// TwinCAT 3 PLC project PLC
// Title: Test
// Company: Gema
// Author: RG
// ProjectVersion: 0.1.0.0
// ProgramVersion: 3.1.4023.0
// libraries:
//   Tc2_EtherCAT, * (Beckhoff Automation GmbH)
//   Tc2_Standard, * (Beckhoff Automation GmbH)
//   Tc2_System, * (Beckhoff Automation GmbH)
//   Tc3_Module, * (Beckhoff Automation GmbH)
//   TcoCore, 0.11.0.15 (Vortex.Library)
//   TcoData, 0.11.0.15 (Vortex.Library)
//   TcoDrivesBeckhoff, 0.11.0.15 (Vortex.Library)
//   TcoElements, 0.11.0.15 (Vortex.Library)
//   TcoPneumatics, 0.11.0.15 (Vortex.Library)
//   Vision.Library, * (Gema Technik)
//   BASIC,3.31,OSCAT
// project tree:
//   / PlcTask.TcTTO (not stored)
//   POUs/ AppContext.TcPOU (not stored), MAIN.TcPOU (not stored), MainStation.TcPOU
// real-time tasks:
//   TASK PlcTask: cycle T#1ms, priority 20, ADS port 350
// I/O:
//   DEVICE Device 2 (EtherCAT), AmsNetId 192.168.1.8.3.1
//     Box 1 (DL-EC1A) [DL-EC1A]
// variable links:
//   PLC/PLC Instance <-> Device 2 (EtherCAT)/Box 1 (DL-EC1A)
//     PlcTask Inputs/MAIN._app._mainStation._IvController.ID01 <-> ID01 Current Value  TxPDOMap/ID01 Current Value (P.V.)
//     PlcTask Inputs/MAIN._app._mainStation._IvController.ID01Status @bit 9 <-> ID01 Status TxPDOMap/ID01 Current Value Invalid
//     PlcTask Inputs/MAIN._app._mainStation._IvController.ID02Status @bit 9 <-> ID02 Status TxPDOMap/ID02 Current Value Invalid
//     PlcTask Inputs/MAIN._app._mainStation._IvController.ID03Status @bit 9 <-> ID03 Status TxPDOMap/ID03 Current Value Invalid
//     PlcTask Inputs/MAIN._app._mainStation._IvController.ID04Status @bit 9 <-> ID04 Status TxPDOMap/ID04 Current Value Invalid
//     PlcTask Inputs/MAIN._app._mainStation._IvController.ID05Status @bit 9 <-> ID05 Status TxPDOMap/ID05 Current Value Invalid
//     PlcTask Inputs/MAIN._app._mainStation._IvController.ID06Status @bit 9 <-> ID06 Status TxPDOMap/ID06 Current Value Invalid
//     PlcTask Inputs/MAIN._app._mainStation._IvController.ID07Status @bit 9 <-> ID07 Status TxPDOMap/ID07 Current Value Invalid
//     PlcTask Inputs/MAIN._app._mainStation._IvController.ID08Status @bit 9 <-> ID08 Status TxPDOMap/ID08 Current Value Invalid
//     PlcTask Inputs/MAIN._app._mainStation._IvController.ID01Status @bit 11 <-> ID01 Status TxPDOMap/ID01 Current Value Over Range
//     PlcTask Inputs/MAIN._app._mainStation._IvController.ID02Status @bit 11 <-> ID02 Status TxPDOMap/ID02 Current Value Over Range
//     PlcTask Inputs/MAIN._app._mainStation._IvController.ID03Status @bit 11 <-> ID03 Status TxPDOMap/ID03 Current Value Over Range
//     PlcTask Inputs/MAIN._app._mainStation._IvController.ID04Status @bit 11 <-> ID04 Status TxPDOMap/ID04 Current Value Over Range
//     PlcTask Inputs/MAIN._app._mainStation._IvController.ID05Status @bit 11 <-> ID05 Status TxPDOMap/ID05 Current Value Over Range
//     PlcTask Inputs/MAIN._app._mainStation._IvController.ID06Status @bit 11 <-> ID06 Status TxPDOMap/ID06 Current Value Over Range
//     PlcTask Inputs/MAIN._app._mainStation._IvController.ID07Status @bit 11 <-> ID07 Status TxPDOMap/ID07 Current Value Over Range
//     PlcTask Inputs/MAIN._app._mainStation._IvController.ID08Status @bit 11 <-> ID08 Status TxPDOMap/ID08 Current Value Over Range
//     PlcTask Inputs/MAIN._app._mainStation._IvController.ID01Status @bit 10 <-> ID01 Status TxPDOMap/ID01 Current Value Under Range
//     PlcTask Inputs/MAIN._app._mainStation._IvController.ID02Status @bit 10 <-> ID02 Status TxPDOMap/ID02 Current Value Under Range
//     PlcTask Inputs/MAIN._app._mainStation._IvController.ID03Status @bit 10 <-> ID03 Status TxPDOMap/ID03 Current Value Under Range
//     PlcTask Inputs/MAIN._app._mainStation._IvController.ID04Status @bit 10 <-> ID04 Status TxPDOMap/ID04 Current Value Under Range
//     PlcTask Inputs/MAIN._app._mainStation._IvController.ID05Status @bit 10 <-> ID05 Status TxPDOMap/ID05 Current Value Under Range
//     PlcTask Inputs/MAIN._app._mainStation._IvController.ID06Status @bit 10 <-> ID06 Status TxPDOMap/ID06 Current Value Under Range
//     PlcTask Inputs/MAIN._app._mainStation._IvController.ID07Status @bit 10 <-> ID07 Status TxPDOMap/ID07 Current Value Under Range
//     PlcTask Inputs/MAIN._app._mainStation._IvController.ID08Status @bit 10 <-> ID08 Status TxPDOMap/ID08 Current Value Under Range
//     PlcTask Inputs/MAIN._app._mainStation._IvController.ID01Status @bit 15 <-> ID01 Status TxPDOMap/ID01 Error Status
//     PlcTask Inputs/MAIN._app._mainStation._IvController.ID02Status @bit 15 <-> ID02 Status TxPDOMap/ID02 Error Status
//     PlcTask Inputs/MAIN._app._mainStation._IvController.ID03Status @bit 15 <-> ID03 Status TxPDOMap/ID03 Error Status
//     PlcTask Inputs/MAIN._app._mainStation._IvController.ID04Status @bit 15 <-> ID04 Status TxPDOMap/ID04 Error Status
//     PlcTask Inputs/MAIN._app._mainStation._IvController.ID05Status @bit 15 <-> ID05 Status TxPDOMap/ID05 Error Status
//     PlcTask Inputs/MAIN._app._mainStation._IvController.ID06Status @bit 15 <-> ID06 Status TxPDOMap/ID06 Error Status
//     PlcTask Inputs/MAIN._app._mainStation._IvController.ID07Status @bit 15 <-> ID07 Status TxPDOMap/ID07 Error Status
//     PlcTask Inputs/MAIN._app._mainStation._IvController.ID08Status @bit 15 <-> ID08 Status TxPDOMap/ID08 Error Status
//     PlcTask Inputs/MAIN._app._mainStation._IvController.ID01Status <-> ID01 Status TxPDOMap/ID01 Output 1
//     PlcTask Inputs/MAIN._app._mainStation._IvController.ID02Status <-> ID02 Status TxPDOMap/ID02 Output 1
//     PlcTask Inputs/MAIN._app._mainStation._IvController.ID03Status <-> ID03 Status TxPDOMap/ID03 Output 1
//     PlcTask Inputs/MAIN._app._mainStation._IvController.ID04Status <-> ID04 Status TxPDOMap/ID04 Output 1
//     PlcTask Inputs/MAIN._app._mainStation._IvController.ID05Status <-> ID05 Status TxPDOMap/ID05 Output 1
//     PlcTask Inputs/MAIN._app._mainStation._IvController.ID06Status <-> ID06 Status TxPDOMap/ID06 Output 1
//     PlcTask Inputs/MAIN._app._mainStation._IvController.ID07Status <-> ID07 Status TxPDOMap/ID07 Output 1
//     PlcTask Inputs/MAIN._app._mainStation._IvController.ID08Status <-> ID08 Status TxPDOMap/ID08 Output 1
//     PlcTask Inputs/MAIN._app._mainStation._IvController.ID01Status @bit 1 <-> ID01 Status TxPDOMap/ID01 Output 2
//     PlcTask Inputs/MAIN._app._mainStation._IvController.ID01Status @bit 2 <-> ID01 Status TxPDOMap/ID01 Output 3
//     PlcTask Inputs/MAIN._app._mainStation._IvController.ID01Status @bit 3 <-> ID01 Status TxPDOMap/ID01 Output 4
//     PlcTask Inputs/MAIN._app._mainStation._IvController.ID01Status @bit 4 <-> ID01 Status TxPDOMap/ID01 Output 5
//     PlcTask Inputs/MAIN._app._mainStation._IvController.ID02Status @bit 1 <-> ID02 Status TxPDOMap/ID02 Output 2
//     PlcTask Inputs/MAIN._app._mainStation._IvController.ID02Status @bit 2 <-> ID02 Status TxPDOMap/ID02 Output 3
//     PlcTask Inputs/MAIN._app._mainStation._IvController.ID02Status @bit 3 <-> ID02 Status TxPDOMap/ID02 Output 4
//     PlcTask Inputs/MAIN._app._mainStation._IvController.ID02Status @bit 4 <-> ID02 Status TxPDOMap/ID02 Output 5
//     PlcTask Inputs/MAIN._app._mainStation._IvController.ID03Status @bit 1 <-> ID03 Status TxPDOMap/ID03 Output 2
//     PlcTask Inputs/MAIN._app._mainStation._IvController.ID03Status @bit 2 <-> ID03 Status TxPDOMap/ID03 Output 3
//     PlcTask Inputs/MAIN._app._mainStation._IvController.ID03Status @bit 3 <-> ID03 Status TxPDOMap/ID03 Output 4
//     PlcTask Inputs/MAIN._app._mainStation._IvController.ID03Status @bit 4 <-> ID03 Status TxPDOMap/ID03 Output 5
//     PlcTask Inputs/MAIN._app._mainStation._IvController.ID04Status @bit 1 <-> ID04 Status TxPDOMap/ID04 Output 2
//     PlcTask Inputs/MAIN._app._mainStation._IvController.ID04Status @bit 2 <-> ID04 Status TxPDOMap/ID04 Output 3
//     PlcTask Inputs/MAIN._app._mainStation._IvController.ID04Status @bit 3 <-> ID04 Status TxPDOMap/ID04 Output 4
//     PlcTask Inputs/MAIN._app._mainStation._IvController.ID04Status @bit 4 <-> ID04 Status TxPDOMap/ID04 Output 5
//     PlcTask Inputs/MAIN._app._mainStation._IvController.ID05Status @bit 1 <-> ID05 Status TxPDOMap/ID05 Output 2
//     PlcTask Inputs/MAIN._app._mainStation._IvController.ID05Status @bit 2 <-> ID05 Status TxPDOMap/ID05 Output 3
//     PlcTask Inputs/MAIN._app._mainStation._IvController.ID05Status @bit 3 <-> ID05 Status TxPDOMap/ID05 Output 4
//     PlcTask Inputs/MAIN._app._mainStation._IvController.ID05Status @bit 4 <-> ID05 Status TxPDOMap/ID05 Output 5
//     PlcTask Inputs/MAIN._app._mainStation._IvController.ID06Status @bit 1 <-> ID06 Status TxPDOMap/ID06 Output 2
//     PlcTask Inputs/MAIN._app._mainStation._IvController.ID06Status @bit 2 <-> ID06 Status TxPDOMap/ID06 Output 3
//     PlcTask Inputs/MAIN._app._mainStation._IvController.ID06Status @bit 3 <-> ID06 Status TxPDOMap/ID06 Output 4
//     PlcTask Inputs/MAIN._app._mainStation._IvController.ID06Status @bit 4 <-> ID06 Status TxPDOMap/ID06 Output 5
//     PlcTask Inputs/MAIN._app._mainStation._IvController.ID07Status @bit 1 <-> ID07 Status TxPDOMap/ID07 Output 2
//     PlcTask Inputs/MAIN._app._mainStation._IvController.ID07Status @bit 2 <-> ID07 Status TxPDOMap/ID07 Output 3
//     PlcTask Inputs/MAIN._app._mainStation._IvController.ID07Status @bit 3 <-> ID07 Status TxPDOMap/ID07 Output 4
//     PlcTask Inputs/MAIN._app._mainStation._IvController.ID07Status @bit 4 <-> ID07 Status TxPDOMap/ID07 Output 5
//     PlcTask Inputs/MAIN._app._mainStation._IvController.ID08Status @bit 1 <-> ID08 Status TxPDOMap/ID08 Output 2
//     PlcTask Inputs/MAIN._app._mainStation._IvController.ID08Status @bit 2 <-> ID08 Status TxPDOMap/ID08 Output 3
//     PlcTask Inputs/MAIN._app._mainStation._IvController.ID08Status @bit 3 <-> ID08 Status TxPDOMap/ID08 Output 4
//     PlcTask Inputs/MAIN._app._mainStation._IvController.ID08Status @bit 4 <-> ID08 Status TxPDOMap/ID08 Output 5
//     PlcTask Inputs/MAIN._app._mainStation._IvController.ID01Status @bit 14 <-> ID01 Status TxPDOMap/ID01 Warning Status
//     PlcTask Inputs/MAIN._app._mainStation._IvController.ID02Status @bit 14 <-> ID02 Status TxPDOMap/ID02 Warning Status
//     PlcTask Inputs/MAIN._app._mainStation._IvController.ID03Status @bit 14 <-> ID03 Status TxPDOMap/ID03 Warning Status
//     PlcTask Inputs/MAIN._app._mainStation._IvController.ID04Status @bit 14 <-> ID04 Status TxPDOMap/ID04 Warning Status
//     PlcTask Inputs/MAIN._app._mainStation._IvController.ID05Status @bit 14 <-> ID05 Status TxPDOMap/ID05 Warning Status
//     PlcTask Inputs/MAIN._app._mainStation._IvController.ID06Status @bit 14 <-> ID06 Status TxPDOMap/ID06 Warning Status
//     PlcTask Inputs/MAIN._app._mainStation._IvController.ID07Status @bit 14 <-> ID07 Status TxPDOMap/ID07 Warning Status
//     PlcTask Inputs/MAIN._app._mainStation._IvController.ID08Status @bit 14 <-> ID08 Status TxPDOMap/ID08 Warning Status
//     PlcTask Inputs/MAIN._app._mainStation._IvController.ID01Status @bit 5 <-> ID01 Status TxPDOMap/Reserved
//     PlcTask Inputs/MAIN._app._mainStation._IvController.ID02Status @bit 5 <-> ID02 Status TxPDOMap/Reserved
//     PlcTask Inputs/MAIN._app._mainStation._IvController.ID03Status @bit 5 <-> ID03 Status TxPDOMap/Reserved
//     PlcTask Inputs/MAIN._app._mainStation._IvController.ID04Status @bit 5 <-> ID04 Status TxPDOMap/Reserved
//     PlcTask Inputs/MAIN._app._mainStation._IvController.ID05Status @bit 5 <-> ID05 Status TxPDOMap/Reserved
//     PlcTask Inputs/MAIN._app._mainStation._IvController.ID06Status @bit 5 <-> ID06 Status TxPDOMap/Reserved
//     PlcTask Inputs/MAIN._app._mainStation._IvController.ID07Status @bit 5 <-> ID07 Status TxPDOMap/Reserved
//     PlcTask Inputs/MAIN._app._mainStation._IvController.ID08Status @bit 5 <-> ID08 Status TxPDOMap/Reserved
//     PlcTask Inputs/MAIN._app._mainStation._IvController.ID01Status @bit 6 <-> ID01 Status TxPDOMap/Reserved_1
//     PlcTask Inputs/MAIN._app._mainStation._IvController.ID01Status @bit 7 <-> ID01 Status TxPDOMap/Reserved_2
//     PlcTask Inputs/MAIN._app._mainStation._IvController.ID01Status @bit 8 <-> ID01 Status TxPDOMap/Reserved_3
//     PlcTask Inputs/MAIN._app._mainStation._IvController.ID01Status @bit 12 <-> ID01 Status TxPDOMap/Reserved_4
//     PlcTask Inputs/MAIN._app._mainStation._IvController.ID01Status @bit 13 <-> ID01 Status TxPDOMap/Reserved_5
//     PlcTask Inputs/MAIN._app._mainStation._IvController.ID02Status @bit 6 <-> ID02 Status TxPDOMap/Reserved_1
//     PlcTask Inputs/MAIN._app._mainStation._IvController.ID02Status @bit 7 <-> ID02 Status TxPDOMap/Reserved_2
//     PlcTask Inputs/MAIN._app._mainStation._IvController.ID02Status @bit 8 <-> ID02 Status TxPDOMap/Reserved_3
//     PlcTask Inputs/MAIN._app._mainStation._IvController.ID02Status @bit 12 <-> ID02 Status TxPDOMap/Reserved_4
//     PlcTask Inputs/MAIN._app._mainStation._IvController.ID02Status @bit 13 <-> ID02 Status TxPDOMap/Reserved_5
//     PlcTask Inputs/MAIN._app._mainStation._IvController.ID03Status @bit 6 <-> ID03 Status TxPDOMap/Reserved_1
//     PlcTask Inputs/MAIN._app._mainStation._IvController.ID03Status @bit 7 <-> ID03 Status TxPDOMap/Reserved_2
//     PlcTask Inputs/MAIN._app._mainStation._IvController.ID03Status @bit 8 <-> ID03 Status TxPDOMap/Reserved_3
//     PlcTask Inputs/MAIN._app._mainStation._IvController.ID03Status @bit 12 <-> ID03 Status TxPDOMap/Reserved_4
//     PlcTask Inputs/MAIN._app._mainStation._IvController.ID03Status @bit 13 <-> ID03 Status TxPDOMap/Reserved_5
//     PlcTask Inputs/MAIN._app._mainStation._IvController.ID04Status @bit 6 <-> ID04 Status TxPDOMap/Reserved_1
//     PlcTask Inputs/MAIN._app._mainStation._IvController.ID04Status @bit 7 <-> ID04 Status TxPDOMap/Reserved_2
//     PlcTask Inputs/MAIN._app._mainStation._IvController.ID04Status @bit 8 <-> ID04 Status TxPDOMap/Reserved_3
//     PlcTask Inputs/MAIN._app._mainStation._IvController.ID04Status @bit 12 <-> ID04 Status TxPDOMap/Reserved_4
//     PlcTask Inputs/MAIN._app._mainStation._IvController.ID04Status @bit 13 <-> ID04 Status TxPDOMap/Reserved_5
//     PlcTask Inputs/MAIN._app._mainStation._IvController.ID05Status @bit 6 <-> ID05 Status TxPDOMap/Reserved_1
//     PlcTask Inputs/MAIN._app._mainStation._IvController.ID05Status @bit 7 <-> ID05 Status TxPDOMap/Reserved_2
//     PlcTask Inputs/MAIN._app._mainStation._IvController.ID05Status @bit 8 <-> ID05 Status TxPDOMap/Reserved_3
//     PlcTask Inputs/MAIN._app._mainStation._IvController.ID05Status @bit 12 <-> ID05 Status TxPDOMap/Reserved_4
//     PlcTask Inputs/MAIN._app._mainStation._IvController.ID05Status @bit 13 <-> ID05 Status TxPDOMap/Reserved_5
//     PlcTask Inputs/MAIN._app._mainStation._IvController.ID06Status @bit 6 <-> ID06 Status TxPDOMap/Reserved_1
//     PlcTask Inputs/MAIN._app._mainStation._IvController.ID06Status @bit 7 <-> ID06 Status TxPDOMap/Reserved_2
//     PlcTask Inputs/MAIN._app._mainStation._IvController.ID06Status @bit 8 <-> ID06 Status TxPDOMap/Reserved_3
//     PlcTask Inputs/MAIN._app._mainStation._IvController.ID06Status @bit 12 <-> ID06 Status TxPDOMap/Reserved_4
//     PlcTask Inputs/MAIN._app._mainStation._IvController.ID06Status @bit 13 <-> ID06 Status TxPDOMap/Reserved_5
//     PlcTask Inputs/MAIN._app._mainStation._IvController.ID07Status @bit 6 <-> ID07 Status TxPDOMap/Reserved_1
//     PlcTask Inputs/MAIN._app._mainStation._IvController.ID07Status @bit 7 <-> ID07 Status TxPDOMap/Reserved_2
//     PlcTask Inputs/MAIN._app._mainStation._IvController.ID07Status @bit 8 <-> ID07 Status TxPDOMap/Reserved_3
//     PlcTask Inputs/MAIN._app._mainStation._IvController.ID07Status @bit 12 <-> ID07 Status TxPDOMap/Reserved_4
//     PlcTask Inputs/MAIN._app._mainStation._IvController.ID07Status @bit 13 <-> ID07 Status TxPDOMap/Reserved_5
//     PlcTask Inputs/MAIN._app._mainStation._IvController.ID08Status @bit 6 <-> ID08 Status TxPDOMap/Reserved_1
//     PlcTask Inputs/MAIN._app._mainStation._IvController.ID08Status @bit 7 <-> ID08 Status TxPDOMap/Reserved_2
//     PlcTask Inputs/MAIN._app._mainStation._IvController.ID08Status @bit 8 <-> ID08 Status TxPDOMap/Reserved_3
//     PlcTask Inputs/MAIN._app._mainStation._IvController.ID08Status @bit 12 <-> ID08 Status TxPDOMap/Reserved_4
//     PlcTask Inputs/MAIN._app._mainStation._IvController.ID08Status @bit 13 <-> ID08 Status TxPDOMap/Reserved_5
//     PlcTask Inputs/MAIN._app._mainStation._IvController.ID02_MatchingRateOfPositionAdujustmentTool_01 <-> ID02 Current Value  TxPDOMap/ID02 Current Value (P.V.)
//     PlcTask Inputs/MAIN._app._mainStation._IvController.ID02_MatchingRateOfPositionAdujustmentTool_02 <-> ID03 Current Value  TxPDOMap/ID03 Current Value (P.V.)
//     PlcTask Inputs/MAIN._app._mainStation._IvController.ID02_MatchingRateOfPositionAdujustmentTool_03 <-> ID04 Current Value  TxPDOMap/ID04 Current Value (P.V.)
//     PlcTask Inputs/MAIN._app._mainStation._IvController.ID02_MatchingRateOfPositionAdujustmentTool_04 <-> ID05 Current Value  TxPDOMap/ID05 Current Value (P.V.)
//     PlcTask Inputs/MAIN._app._mainStation._IvController.ID02_MatchingRateOfPositionAdujustmentTool_05 <-> ID06 Current Value  TxPDOMap/ID06 Current Value (P.V.)
//     PlcTask Inputs/MAIN._app._mainStation._IvController.ID02_MatchingRateOfPositionAdujustmentTool_06 <-> ID07 Current Value  TxPDOMap/ID07 Current Value (P.V.)
//     PlcTask Inputs/MAIN._app._mainStation._IvController.ID02_MatchingRateOfPositionAdujustmentTool_07 <-> ID08 Current Value  TxPDOMap/ID08 Current Value (P.V.)
//     PlcTask Inputs/MAIN._app._mainStation._IvController.InfoData/AdsAddr <-> InfoData/AdsAddr
//     PlcTask Inputs/MAIN._app._mainStation._IvController.InfoData/DcInputShift <-> InfoData/DcInputShift
//     PlcTask Inputs/MAIN._app._mainStation._IvController.InfoData/DcOutputShift <-> InfoData/DcOutputShift
//     PlcTask Inputs/MAIN._app._mainStation._IvController.InfoData/State <-> InfoData/State
//     PlcTask Inputs/MAIN._app._mainStation._IvController.InputResponse{1..5} <-> Input Response {1..5} TxPDOMap/Input Response {1..5}  (5 links)
//     PlcTask Inputs/MAIN._app._mainStation._IvController.StatusOfSystem @bit 3 <-> Status of System TxPDOMap/Current Value Property
//     PlcTask Inputs/MAIN._app._mainStation._IvController.StatusOfSystem @bit 16 <-> Status of System TxPDOMap/Error Code
//     PlcTask Inputs/MAIN._app._mainStation._IvController.StatusOfSystem <-> Status of System TxPDOMap/Error Status
//     PlcTask Inputs/MAIN._app._mainStation._IvController.StatusOfSystem @bit 2 <-> Status of System TxPDOMap/Reserved
//     PlcTask Inputs/MAIN._app._mainStation._IvController.StatusOfSystem @bit {4..8} <-> Status of System TxPDOMap/Reserved_{1..5}  (5 links)
//     PlcTask Inputs/MAIN._app._mainStation._IvController.StatusOfSystem @bit 1 <-> Status of System TxPDOMap/Warning Status
//     PlcTask Inputs/MAIN._app._mainStation._IvController.WcState/InputToggle <-> WcState/InputToggle
//     PlcTask Inputs/MAIN._app._mainStation._IvController.WcState/WcState <-> WcState/WcState
//     PlcTask Outputs/MAIN._app._mainStation._IvController.InputRequest{1..5} <-> Input Request {1..5} RxPDOMap/Request {1..5}  (5 links)

// ---- POUs/MainStation.TcPOU
FUNCTION_BLOCK MainStation EXTENDS TcoCore.TcoObject
VAR
    counter : INT;

    _IvController : Vision_Library.IVController(THIS^);
    _trigger      : BOOL;
    _coordinate   : BOOL;
    _coordinates  : ARRAY[0..2] OF Vision_Library.Coordinates;
	_distanceFromObject: LREAL;
END_VAR

counter := counter + 1;

IF (THIS^.counter MOD 13 = 0) THEN
    THIS^.Messenger.Info('opalalla').Pin();
END_IF

IF (THIS^.counter MOD 400 = 0) THEN
    THIS^.Messenger.Error('ich Poste').Pin();
END_IF

_IvController();

IF _trigger THEN
    IF _IvController.TriggerSensorMethod().Done THEN
        _trigger := FALSE;
    end_if
END_IF

IF _coordinate THEN
    IF _IvController.ReadTool1CoordinatesMethod().Done
           and _IvController.ReadTool2CoordinatesMethod().Done
           and _IvController.ReadTool3CoordinatesMethod().Done THEN
        _coordinate     := FALSE;
        _coordinates[0] := _IvController.RawCoordinatesTool1;
        _coordinates[1] := _IvController.RawCoordinatesTool2;
        _coordinates[2] := _IvController.RawCoordinatesTool3;

        _distanceFromObject := _IvController._readTool2CoordinatesTask.DistanceFromObject;
    END_IF
END_IF

END_FUNCTION_BLOCK
